{attribute 'GeneratedUsingTerminal: EL6224-0000-0021'}
{attribute addProperty BoxType "EL6224-0000-0021"}
{attribute addProperty Id "Bitheader_1AT %Q*BYTE1Byte_xAT %Q*ARRAY[0..7] OF BYTE8Bitheader_2AT %Q*BYTE1"}
{attribute addProperty CRC "2855058970"}
{attribute addProperty Size "10"}
TYPE IO_Link_Port2_out_F2E0F4CF EXTENDS OutputBase_10CEE7DE :
STRUCT
	{attribute addProperty Name "Bitheader_1"}
	Bitheader_1 AT %Q* : BYTE;
	{attribute addProperty Name "Byte"}
	Byte_x AT %Q* : ARRAY[0..7] OF BYTE;
	{attribute addProperty Name "Bitheader_2"}
	Bitheader_2 AT %Q* : BYTE;
END_STRUCT
END_TYPE

(* stored: Version 1.2.0.0, ProductVersion 3.1.4024.9
   DUT IO_Link_Port2_out_F2E0F4CF: Id {39d48425-0a40-4fb2-932a-d69cc81fd5c5} *)
